PROGRAM PID_ctrl
VAR
	FB_BasicPID_0: FB_BasicPID;
	Stn3FlowRawData: LREAL;
	Stn3ActualFlowRawData: LREAL;
	bReset: BOOL;
	
	rCtrlCycletime						: REAL 	:= 0.01;
	Stn3_PID_fKp_						: REAL 	:= 1					; (*1.0*)
	Stn3_PID_tTn_						: REAL	:= 1				;
	Stn3_PID_tTv_						: REAL	:= 0.03				;
	Stn3_PID_tTd_						: REAL	:= 0.04				;
	
	
	rPump3_Freq_Reading_Raw: LREAL;
	rPump3_Freq_Reading_Raw_new: LREAL;
	nerrorStatus: UINT;
	rPump3_Freq_Reading_Raw_2: REAL;
	
	
	//PID_FB_0: PID_FB;
	iStn3FlowRawData					: INT;
	iStn3ActualFlowRawData				: INT;
	Stn3_PID_fKp						: REAL := 0.2					; (*1.0*)
	Stn3_PID_tTn						: TIME := T#1S				;
	Stn3_PID_tTv						: TIME := T#30ms				;
	Stn3_PID_tTd						: TIME := T#40MS				;
	

END_VAR

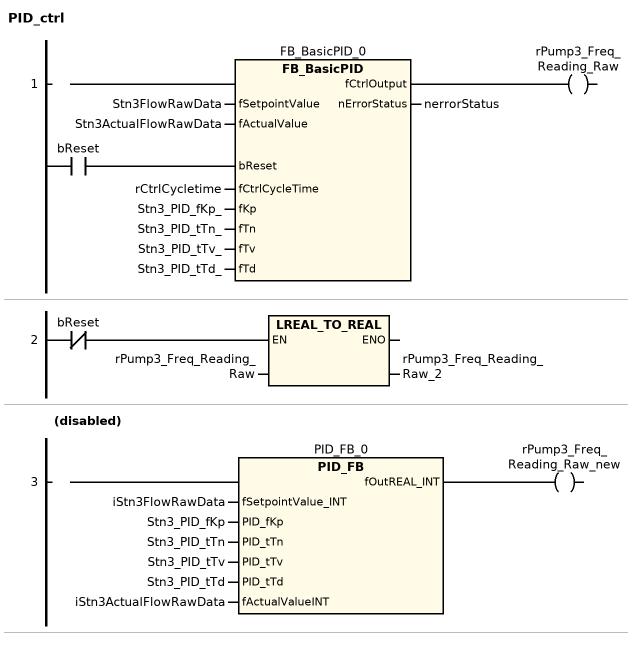
// NETWORK 1
FB_BasicPID_0(
    fSetpointValue := Stn3FlowRawData,
    fActualValue := Stn3ActualFlowRawData,
    bReset := bReset,
    fCtrlCycleTime := rCtrlCycletime,
    fKp := Stn3_PID_fKp_,
    fTn := Stn3_PID_tTn_,
    fTv := Stn3_PID_tTv_,
    fTd := Stn3_PID_tTd_,
    nErrorStatus => nerrorStatus); // FB_BasicPID
rPump3_Freq_Reading_Raw := FB_BasicPID_0.fCtrlOutput;

// NETWORK 2
IF NOT bReset THEN rPump3_Freq_Reading_Raw_2 := LREAL_TO_REAL(rPump3_Freq_Reading_Raw); END_IF

// NETWORK 3 (disabled)
// PID_FB_0(
//     fSetpointValue_INT := iStn3FlowRawData,
//     PID_fKp := Stn3_PID_fKp,
//     PID_tTn := Stn3_PID_tTn,
//     PID_tTv := Stn3_PID_tTv,
//     PID_tTd := Stn3_PID_tTd,
//     fActualValueINT := iStn3ActualFlowRawData); // PID_FB
// rPump3_Freq_Reading_Raw_new := PID_FB_0.fOutREAL_INT;

END_PROGRAM

(* stored: Version 1.1.0.1, ProductVersion 3.1.4024.12
   POU PID_ctrl: Id {606107fc-183d-4f54-b7df-7bc2d2919adb}, SpecialFunc None *)
